Staubli VAL3: allBool.pgx

public program allBool(bool& x_bInput[], bool& x_bResult)
  local num l_nLength
  local num l_nElement
begin

  l_nLength = size(x_bInput)
  x_bResult = false

  for l_nElement = 0 to l_nLength-1
    if x_bInput[l_nElement] == false
      x_bResult = false
      return
    else
      x_bResult = true
    endIf
  endFor

end
